{attribute 'qualified_only'}
VAR_GLOBAL
	controller : Controller;
	joyLeft : LREAL;
END_VAR

(* stored: Version 1.1.0.1, ProductVersion 3.1.4024.9
   GVL XboxControl: Id {4450970d-8615-4fbc-a6f1-cadf92ba8024} *)
